(* PLC project industrial-machine-simulation.project, CODESYS CODESYS V3.5 SP22 Patch 2 *)
(* stored: creationDateTime 2026-10-06T16:26:03.0821542, modificationDateTime 2026-10-06T16:23:11.8509653 *)

{attribute 'do_checks_for_implicit_code'}
PROGRAM PLC_PRG
  VAR
    bBTN_Paro : BOOL;
    siEstados : SINT;
    stEstados : STRING(INT#20);
    bBTN_Home : BOOL;
    bBTN_Manual : BOOL;
    bBTN_Auto : BOOL;
    bIniciarPrograma : BOOL;
    bTestsInicio : BOOL;
  END_VAR
  VAR  (* added by the conversion: wires and edge detectors of the diagram *)
    _MOVE11_EN : BOOL;
    _MOVE19_EN : BOOL;
    _MOVE27_EN : BOOL;
  END_VAR

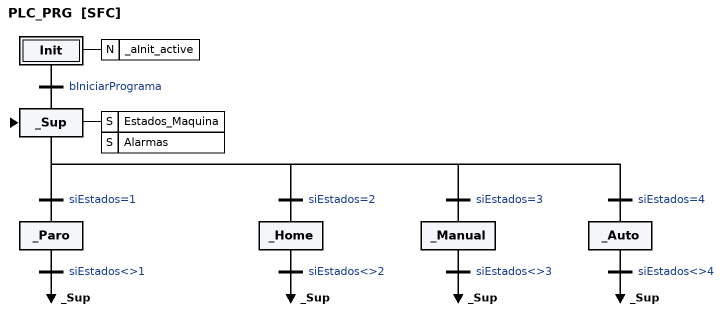
INITIAL_STEP Init:
  _aInit_active(N);
END_STEP
TRANSITION FROM Init TO _Sup
  := bIniciarPrograma;
END_TRANSITION
STEP _Sup:
  Estados_Maquina(S);
  Alarmas(S);
END_STEP
TRANSITION FROM _Sup TO _Paro
  := siEstados=1;
END_TRANSITION
TRANSITION FROM _Sup TO _Home
  := siEstados=2;
END_TRANSITION
TRANSITION FROM _Sup TO _Manual
  := siEstados=3;
END_TRANSITION
TRANSITION FROM _Sup TO _Auto
  := siEstados=4;
END_TRANSITION
STEP _Paro:
END_STEP
TRANSITION FROM _Paro TO _Sup
  := siEstados<>1;
END_TRANSITION
STEP _Home:
END_STEP
TRANSITION FROM _Home TO _Sup
  := siEstados<>2;
END_TRANSITION
STEP _Manual:
END_STEP
TRANSITION FROM _Manual TO _Sup
  := siEstados<>3;
END_TRANSITION
STEP _Auto:
END_STEP
TRANSITION FROM _Auto TO _Sup
  := siEstados<>4;
END_TRANSITION

ACTION Estados_Maquina:
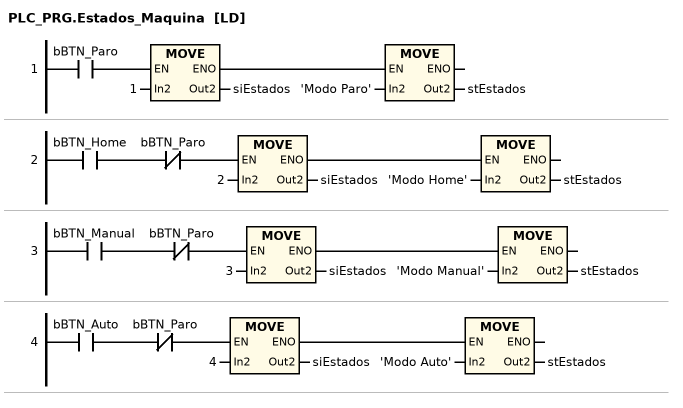
(* LD diagram, written out as Structured Text *)

IF bBTN_Paro THEN siEstados := 1; END_IF;
IF bBTN_Paro THEN stEstados := 'Modo Paro'; END_IF;

_MOVE11_EN := bBTN_Home AND NOT bBTN_Paro;
IF _MOVE11_EN THEN siEstados := 2; END_IF;
IF _MOVE11_EN THEN stEstados := 'Modo Home'; END_IF;

_MOVE19_EN := bBTN_Manual AND NOT bBTN_Paro;
IF _MOVE19_EN THEN siEstados := 3; END_IF;
IF _MOVE19_EN THEN stEstados := 'Modo Manual'; END_IF;

_MOVE27_EN := bBTN_Auto AND NOT bBTN_Paro;
IF _MOVE27_EN THEN siEstados := 4; END_IF;
IF _MOVE27_EN THEN stEstados := 'Modo Auto'; END_IF;
END_ACTION

ACTION Alarmas:
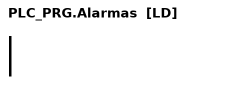
(* LD diagram, written out as Structured Text *)
(* --- network --- *)
END_ACTION

ACTION _aInit_active:
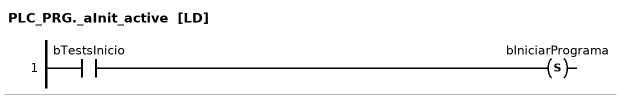
(* LD diagram, written out as Structured Text *)

IF bTestsInicio THEN bIniciarPrograma := TRUE; END_IF;
END_ACTION
END_PROGRAM

PROGRAM SmokeTest

                    GVL.xOutput := GVL.xInput;
                  
END_PROGRAM

CONFIGURATION Device
  RESOURCE Application ON PLC
    {attribute 'qualified_only'}
    VAR_GLOBAL  (* GVL *)
      xInput : BOOL;
      xOutput : BOOL;
    END_VAR
    TASK MainTask(INTERVAL := T#20ms, PRIORITY := 1);
    TASK VISU_TASK(INTERVAL := T#100ms, PRIORITY := 31);
    PROGRAM PLC_PRG WITH MainTask : PLC_PRG;
    PROGRAM SmokeTest WITH MainTask : SmokeTest;
    PROGRAM VisuElems.Visu_Prg WITH VISU_TASK : VisuElems.Visu_Prg;
  END_RESOURCE
END_CONFIGURATION

CONFIGURATION Ethernet
END_CONFIGURATION

CONFIGURATION Modbus_TCP_Client
END_CONFIGURATION

CONFIGURATION Modbus_TCP_Server
END_CONFIGURATION
